FUNCTION_BLOCK FB_PIDControllerConsumer
VAR
    controller : B5PIDController_Plc.FB_PIDController;
    output : REAL;
END_VAR

controller(fError := 2.5);
output := controller.Step();

END_FUNCTION_BLOCK

(* stored: Version 1.1.0.1
   POU FB_PIDControllerConsumer: Id {b9376dec-8586-40c0-9a26-ac7f28a46167}, SpecialFunc None *)
